RoboDK station: URtestcell.rdk

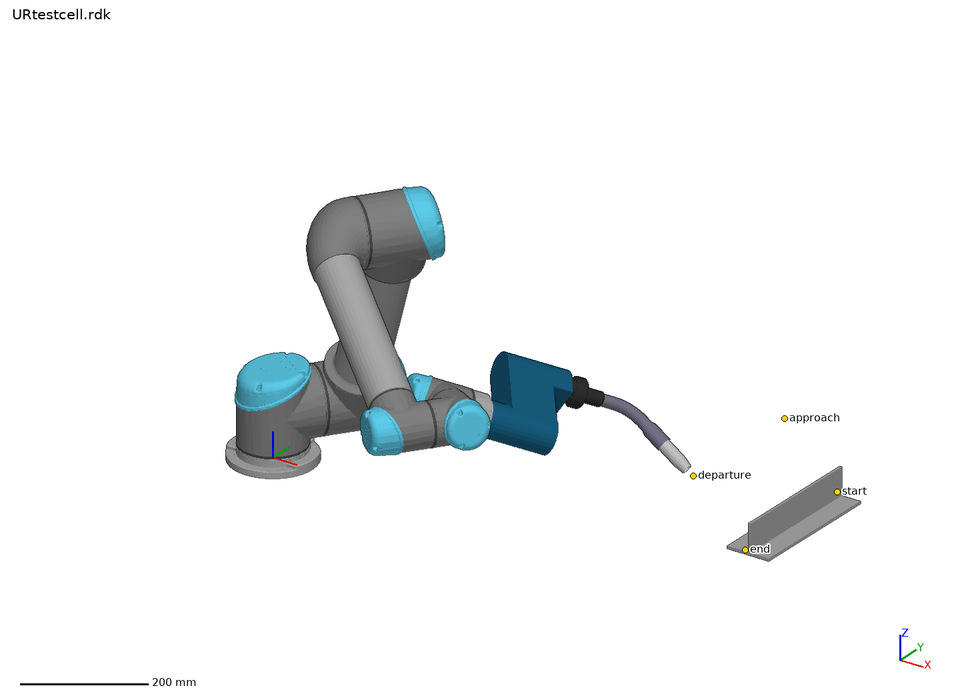
[picture v0: the station drawn from its stored meshes, robots at their saved joint values, targets as dots, program paths as lines]
Station URtestcell (saved by RoboDK 5.8.0). Poses are relative to the parent item; angles as X-Y-Z fixed-axis rotations.
  - frame UR5 Base at (0, 0, 0) mm
    - robot UR5: 6 axes, payload 5 kg, reach 850 mm, repeatability 0.1 mm, weight 18.4 kg
        modified DH rows (alpha deg, a mm, theta deg, d mm): 0, 0, 0, 89.2; 90, 0, 180, 0; 0, 425, 0, 0; 0, 392.43, 0, 109; -90, 0, 0, 93.65; 90, 0, 180, 82
        joint limits [-360, -360, -360, -360, -360, -360] to [360, 360, 360, 360, 360, 360]; home [0, -90, -90, 0, 90, 0]; saved at [144.859, -62.919, 88.158, 55.43, 24.269, -233.441]
      - tool Weld gun, TCP at (-4, 0, 371.3) mm, rotated rx 0 ry 45 rz 0 deg, size 299.9 x 60 x 318.3 mm
    - target approach (Cartesian target) at (695.9, 400, 102.87) mm, rotated rx -125 ry 0 rz -90 deg; joints [144.859, -62.919, 88.158, 55.43, 24.269, -233.441] of UR5
    - target start (Cartesian target) at (795.9, 400, 2.87) mm, rotated rx -125 ry 0 rz -90 deg; joints [144.859, -62.919, 88.158, 55.43, 24.269, -233.441] of UR5
    - target end (Cartesian target) at (795.9, 150, 2.87) mm, rotated rx -125 ry 0 rz -90 deg; joints [144.859, -62.919, 88.158, 55.43, 24.269, -233.441] of UR5
    - target departure (Cartesian target) at (695.9, 150, 102.87) mm, rotated rx -125 ry 0 rz -90 deg; joints [144.859, -62.919, 88.158, 55.43, 24.269, -233.441] of UR5
  - object TJoint A.1 at (800, 400, 0) mm, rotated rx 0 ry -90 rz 90 deg, size 55 x 80 x 250 mm, geometry from TJoint A.1.stl
  - Python program FramesExercise4 (listed below)
  - Python program DemoProgram (listed below)

--- Python program FramesExercise4 ---
from robolink import *    # API to communicate with RoboDK
from robodk import *      # basic matrix operations
import numpy as np


# Any interaction with RoboDK must be done through
# Robolink()
RL = Robolink()

# get the robot item:
robot = RL.Item('UR5 Base',ITEM_TYPE_ROBOT)

#STEP 1:
# jump to a location Set the home joints
jhome = [ 150, -110, 100, 30, 70, -50];

# Set the robot at the home position
robot.MoveJ(jhome);


# Make locations

bTe=transl(800,400,00)*rotz(90*pi/180)*roty(-90*pi/180)


# transformations from {E} to tool (note it is the tool as defided in the
# exercise)


v = 35*pi/180;
s = 5;
L = 250;

eTtoolstart=Mat([[-cos(v), -sin(v), 0, s*sin(v)],
                [ sin(v), -cos(v), 0,  s*cos(v)],
                [  0    , 0      , 1,    0    ],
                [  0    , 0      , 0,    1    ]])

eTtoolend  =Mat([[-cos(v), -sin(v), 0, s*sin(v)],
                [ sin(v), -cos(v), 0,  s*cos(v)],
                [  0    , 0      , 1,    L    ],
                [  0    , 0      , 0,    1    ]])


eTtoolapproach =Mat([[-cos(v), -sin(v), 0, s*sin(v)+100],
                    [ sin(v), -cos(v), 0,  s*cos(v)+100],
                    [  0    , 0      , 1,    0    ],
                    [  0    , 0      , 0,    1    ]])


eTtooldepart =Mat([[-cos(v), -sin(v), 0, s*sin(v)+100],
                    [ sin(v), -cos(v), 0,  s*cos(v)+100],
                    [  0    , 0      , 1,    L    ],
                    [  0    , 0      , 0,    1    ]])

# transformations from Tool in exercise to tool in RoboDK

toolTtoolrobot=Mat([[0, 1, 0, 0],
                    [0, 0, 1, 0],
                    [1, 0, 0, 0],
                    [0, 0, 0, 1]])

# Lets compute the desired locations
bTapproach=bTe*eTtoolapproach*toolTtoolrobot
bTstart   =bTe*eTtoolstart*toolTtoolrobot
bTend     =bTe*eTtoolend*toolTtoolrobot
bTdepart  =bTe*eTtooldepart*toolTtoolrobot

# lets test the movements

robot.MoveL(bTapproach);
robot.MoveL(bTstart);
robot.MoveL(bTend);
robot.MoveL(bTdepart);

## Lets make a program
prog = RL.AddProgram('My program');

target = RL.AddTarget('approach');
target.setPose(bTapproach);
prog.MoveL(target);

target = RL.AddTarget('start');
target.setPose(bTstart);
prog.MoveL(target);

target = RL.AddTarget('end');
target.setPose(bTend);
prog.MoveL(target);

target = RL.AddTarget('departure');
target.setPose(bTdepart);
prog.MoveL(target);

--- Python program DemoProgram ---
# Type help("robolink") or help("robodk") for more information
# Press F5 to run the script
# Documentation: https://robodk.com/doc/en/RoboDK-API.html
# Reference:     https://robodk.com/doc/en/PythonAPI/index.html
# Note: It is not required to keep a copy of this file, your python script is saved with the station
from robolink import *    # RoboDK API
from robodk import *      # Robot toolbox
RDK = Robolink()

# Select a robot (popup is displayed if more than one robot is available)
robot = RDK.ItemUserPick('Select a robot', ITEM_TYPE_ROBOT)
if not robot.Valid():
    raise Exception('No robot selected or available')

# get the current position of the TCP with respect to the reference frame:
# (4x4 matrix representing position and orientation)
target_ref = robot.Pose()
pos_ref = target_ref.Pos()
print("Drawing a polygon around the target: ")
print(Pose_2_TxyzRxyz(target_ref))

# move the robot to the first point:
robot.MoveJ(target_ref)

# It is important to provide the reference frame and the tool frames when generating programs offline
robot.setPoseFrame(robot.PoseFrame())
robot.setPoseTool(robot.PoseTool())
robot.setRounding(10)  # Set the rounding parameter (Also known as: CNT, APO/C_DIS, ZoneData, Blending radius, cornering, ...)
robot.setSpeed(200)  # Set linear speed in mm/s

# Set the number of sides of the polygon:
n_sides = 6
R = 100

# make a hexagon around reference target:
for i in range(n_sides + 1):
    ang = i * 2 * pi / n_sides  #angle: 0, 60, 120, ...

    #-----------------------------
    # Movement relative to the reference frame
    # Create a copy of the target
    target_i = Mat(target_ref)
    pos_i = target_i.Pos()
    pos_i[0] = pos_i[0] + R * cos(ang)
    pos_i[1] = pos_i[1] + R * sin(ang)
    target_i.setPos(pos_i)
    print("Moving to target %i: angle %.1f" % (i, ang * 180 / pi))
    print(str(Pose_2_TxyzRxyz(target_i)))
    robot.MoveL(target_i)

    #-----------------------------
    # Post multiply: relative to the tool
    #target_i = target_ref * rotz(ang) * transl(R,0,0) * rotz(-ang)
    #robot.MoveL(target_i)

# move back to the center, then home:
robot.MoveL(target_ref)

print('Done')
